# EPICS autosave request: ADADSC/adscApp/Db/adsc_settings.req
$(P)$(R)ADSCReadConditn.SCAN
$(P)$(R)ADSCReusDrk
$(P)$(R)ADSCDezingr
$(P)$(R)ADSCAdc
$(P)$(R)ADSCRaw
$(P)$(R)ADSCImXform
$(P)$(R)ADSCStrDrks
$(P)$(R)ADSCBeamX
$(P)$(R)ADSCBeamY
$(P)$(R)ADSCDistnce
$(P)$(R)ADSC2Theta
$(P)$(R)ADSCAxis
$(P)$(R)ADSCWavelen
$(P)$(R)ADSCImWidth
$(P)$(R)ADSCPhi
$(P)$(R)ADSCOmega
$(P)$(R)ADSCKappa
file "ADBase_settings.req", P=$(P), R=$(R)
file "NDFile_settings.req", P=$(P), R=$(R)
